// Interface for a set implemented using a hash table.
INTERFACE I_Hash_Set EXTENDS I_Set

// Number of buckets in the hash set.
PROPERTY _Bucket_Count : T_Capacity;
GET
END_GET
END_PROPERTY

// Sets the number of buckets in the hash set.
// Existing items are rehashed and redistributed into the new buckets.
METHOD Resize : I_Hash_Set
VAR_INPUT
	Count : T_Capacity;
END_VAR
END_METHOD

END_INTERFACE

(* stored: Version 1.1.0.1
   Itf I_Hash_Set: Id {7dbde015-f691-0032-105f-319d360a647c}
   Property _Bucket_Count: Id {b499cc5c-2ea2-0e91-22bc-dc4730b1eba3}
   Get Get: Id {63098bce-62be-08ef-1e01-c55123fbd835}
   Method Resize: Id {dc4ea629-bc7c-039b-3b42-57de132f44c5} *)
